RESOURCE_TYPE _Core402
  (* Standard: 61499-2 *)
  (* Version 0.1, 2017-00-01, hpea485, UOA *)
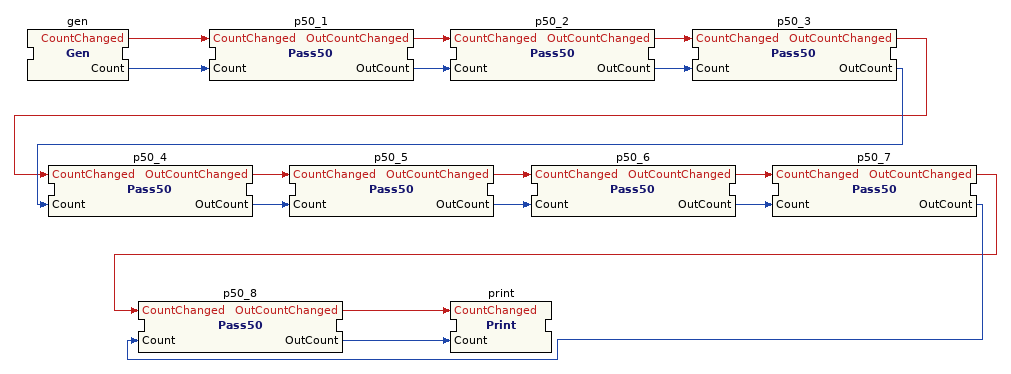
  FBS
    gen : Gen;
    p50_2 : Pass50;
    print : Print;
    p50_1 : Pass50;
    p50_3 : Pass50;
    p50_5 : Pass50;
    p50_4 : Pass50;
    p50_6 : Pass50;
    p50_7 : Pass50;
    p50_8 : Pass50;
  END_FBS
  EVENT_CONNECTIONS
    gen.CountChanged TO p50_1.CountChanged;
    p50_2.OutCountChanged TO p50_3.CountChanged;
    p50_1.OutCountChanged TO p50_2.CountChanged;
    p50_3.OutCountChanged TO p50_4.CountChanged;
    p50_5.OutCountChanged TO p50_6.CountChanged;
    p50_4.OutCountChanged TO p50_5.CountChanged;
    p50_6.OutCountChanged TO p50_7.CountChanged;
    p50_7.OutCountChanged TO p50_8.CountChanged;
    p50_8.OutCountChanged TO print.CountChanged;
  END_CONNECTIONS
  DATA_CONNECTIONS
    gen.Count TO p50_1.Count;
    p50_2.OutCount TO p50_3.Count;
    p50_1.OutCount TO p50_2.Count;
    p50_3.OutCount TO p50_4.Count;
    p50_5.OutCount TO p50_6.Count;
    p50_4.OutCount TO p50_5.Count;
    p50_6.OutCount TO p50_7.Count;
    p50_7.OutCount TO p50_8.Count;
    p50_8.OutCount TO print.Count;
  END_CONNECTIONS
END_RESOURCE_TYPE
